(* IEC 61131-3 sources: Livny/, 3 files *)

(* ---- 03_FB_InputHandler.st ---- *)
(* =========================================================================
   ПРОЕКТ    : Весовой дозатор сахара в мешки 25/50 кг («Ливны»)
   ПЛАТФОРМА : ОВЕН СПК107 · CODESYS 3.5.17 · IEC 61131-3 (Structured Text)
   =========================================================================
   ФАЙЛ      : 03_FB_InputHandler.st
   НАЗНАЧЕНИЕ: Антидребезг дискретных входов (МВ110-8Д.4Р) и выделение
               фронтов кнопок. Дискретизация опроса модуля по RS-485 —
               десятки мс, поэтому фильтруем 40 мс (TON).

               В CODESYS: "Добавить объект → ФБ", язык ST.
   ========================================================================= *)

FUNCTION_BLOCK FB_InputHandler

VAR_INPUT
    xRawStart       : BOOL;   (* «сырой» DI0 ПУСК                         *)
    xRawStop        : BOOL;   (* «сырой» DI1 СТОП                         *)
    xRawEStop       : BOOL;   (* «сырой» DI2 АВАРИЙНЫЙ СТОП (НЗ-контакт)  *)
    xRawBag         : BOOL;   (* «сырой» DI3 мешок в зоне                 *)
    xRawClampClosed : BOOL;   (* «сырой» DI4 концевик зажима              *)
    xRawAirOK       : BOOL;   (* «сырой» DI5 давление воздуха             *)
    xRawLevel       : BOOL;   (* «сырой» DI6 уровень в бункере            *)
    xRawCover       : BOOL;   (* «сырой» DI7 защитная крышка              *)
END_VAR

VAR_OUTPUT
    xStart        : BOOL;     (* ПУСК, отфильтрованный                    *)
    xStop         : BOOL;     (* СТОП, отфильтрованный                    *)
    xStartUp      : BOOL;     (* фронт кнопки ПУСК (один скан)            *)
    xStopUp       : BOOL;     (* фронт кнопки СТОП (один скан)            *)
    xEStop        : BOOL;     (* АВАРИЯ активна (инверсия НЗ-контакта)    *)
    xBagPresent   : BOOL;     (* мешок установлен в зону загрузки         *)
    xClampClosed  : BOOL;     (* зажим механически закрыт                 *)
    xAirOK        : BOOL;     (* давление пневмосети в норме              *)
    xLevelOK      : BOOL;     (* продукт в бункере есть                   *)
    xCoverClosed  : BOOL;     (* защитная крышка закрыта                  *)
END_VAR

VAR
    (* Фильтры антидребезга: TON с выдержкой tDebounce                  *)
    tonStart : TON;
    tonStop  : TON;
    tonEStop : TON;
    tonBag   : TON;
    tonClamp : TON;
    tonAir   : TON;
    tonLevel : TON;
    tonCover : TON;

    (* Детекторы фронта для кнопок                                      *)
    rtStart  : R_TRIG;
    rtStop   : R_TRIG;

    tDebounce : TIME := T#40MS;  (* Постоянная антидребезга               *)
END_VAR

(* ---------------------------------------------------------------------
   1. АНТИДРЕБЕЗГ. Вход считается принятым, если удерживается
      не менее tDebounce. Для цепей безопасности (аварийный стоп)
      это не ухудшает быстродействие: НЗ-контакт при срабатывании
      РАЗМЫКАЕТСЯ, и инверсный признак аварии снимает разрешение
      выходов уже в следующем скане.
   --------------------------------------------------------------------- *)
tonStart(IN := xRawStart,       PT := tDebounce);
tonStop (IN := xRawStop,        PT := tDebounce);
tonEStop(IN := xRawEStop,       PT := tDebounce);
tonBag  (IN := xRawBag,         PT := tDebounce);
tonClamp(IN := xRawClampClosed, PT := tDebounce);
tonAir  (IN := xRawAirOK,       PT := tDebounce);
tonLevel(IN := xRawLevel,       PT := tDebounce);
tonCover(IN := xRawCover,       PT := tDebounce);

xStart       := tonStart.Q;
xStop        := tonStop.Q;

(* Аварийный стоп — НЗ-контакт: пока цепь цела, вход = TRUE.
   Размыкание (нажатие/обрыв) даёт xEStop = TRUE.                     *)
xEStop       := NOT tonEStop.Q;

xBagPresent  := tonBag.Q;
xClampClosed := tonClamp.Q;
xAirOK       := tonAir.Q;
xLevelOK     := tonLevel.Q;
xCoverClosed := tonCover.Q;

(* ---------------------------------------------------------------------
   2. ФРОНТЫ КНОПОК — для запуска/останова цикла из любого состояния.
   --------------------------------------------------------------------- *)
rtStart(CLK := xStart);
xStartUp := rtStart.Q;

rtStop(CLK := xStop);
xStopUp  := rtStop.Q;

END_FUNCTION_BLOCK

(* =========================================================================
   КОНЕЦ ФАЙЛА 03_FB_InputHandler.st
   ========================================================================= *)

(* ---- 05_FB_DoserControl.st ---- *)
(* =========================================================================
   ПРОЕКТ    : Весовой дозатор сахара в мешки 25/50 кг («Ливны»)
   ПЛАТФОРМА : ОВЕН СПК107 · CODESYS 3.5.17 · IEC 61131-3 (Structured Text)
   =========================================================================
   ФАЙЛ      : 05_FB_DoserControl.st
   НАЗНАЧЕНИЕ: Управляющий автомат дозатора (ядро проекта).

   ЦИКЛ ДОЗИРОВАНИЯ:
     ГОТОВНОСТЬ → ЗАЖИМ → ТАРА → ГРУБАЯ ПОДАЧА → ТОЧНАЯ ПОДАЧА →
     УСПОКОЕНИЕ → КОНТРОЛЬ (→ ДОСЫПКА) → СБРОС МЕШКА → ПАУЗА → ГОТОВНОСТЬ

   КЛЮЧЕВЫЕ ПРИНЦИПЫ:
     1. Двухступенчатая подача: основной шнек даёт ~90 % дозы,
        малый шнек — доводка. Это главный способ получить точность
        ±50 г на мешке 25 кг при грубой пневматике/механике.
     2. Отсечка «на лету» (in-flight): питатель закрывается ДО
        достижения уставки на величину продукта, который ещё летит
        в мешок:  W_отс = W_зад − Δ_лету.
     3. Адаптация Δ_лету по ошибке каждой отвешенной дозы:
        ε = W_факт − W_зад ≈ Δ_факт − Δ_принято
        Δ_лету := clamp( Δ_лету + K·ε ,  Δ_min … Δ_max )
     4. Контроль потока: за окно tFlowCheck вес обязан вырасти
        не менее чем на rFlowMinStep — иначе «затор/пусто».
     5. Failsafe: при любой аварии выходы гасятся в том же скане.
   ========================================================================= *)

FUNCTION_BLOCK FB_DoserControl

VAR_INPUT
    xEnable      : BOOL;   (* разрешение работы автоматики               *)
    xAlarmActive : BOOL;   (* есть квитируемые аварии (от FB_AlarmManager)*)
    xStartCmd    : BOOL;   (* импульс «ПУСК» (один скан)                 *)
    xStopCmd     : BOOL;   (* импульс «СТОП» (один скан)                 *)
    xAckCmd      : BOOL;   (* импульс квитирования                       *)

    (* Весовой канал (после FB_WeightChannel)                           *)
    rNet     : REAL;       (* вес нетто, кг                              *)
    xStable  : BOOL;       (* вес стабилен                               *)
    xCommOK  : BOOL;       (* связь с тензомодулем в норме               *)

    (* Дискретные сигналы (после FB_InputHandler)                       *)
    xBagPresent   : BOOL;  (* мешок в зоне загрузки                      *)
    xClampClosed  : BOOL;  (* концевик: зажим закрыт                     *)
    xAirOK        : BOOL;  (* давление пневмосети в норме                *)
    xLevelOK      : BOOL;  (* сахар в расходном бункере есть             *)
    xCoverClosed  : BOOL;  (* защитная крышка закрыта                    *)
    xEStop        : BOOL;  (* аварийный стоп (НЗ-цепь)                   *)

    (* Технологические параметры                                        *)
    p : ST_DoseParams;
END_VAR

VAR_OUTPUT
    xDoClamp  : BOOL;      (* пневмоклапан зажима мешка                  *)
    xDoCoarse : BOOL;      (* грубый питатель (основной шнек)            *)
    xDoFine   : BOOL;      (* точный питатель (малый шнек)               *)
    xTareReq  : BOOL;      (* импульс тарирования → FB_WeightChannel     *)

    eState    : E_DoserState;   (* текущее состояние (для HMI/архива)    *)
    rInFlight : REAL;           (* текущая адаптивная отсечка, кг        *)
    rLastError: REAL;           (* ошибка последней дозы, кг             *)

    (* Запросы на аварии (защёлкиваются в FB_AlarmManager)              *)
    xReqTareFault : BOOL;
    xReqNoFlow    : BOOL;
    xReqOverdose  : BOOL;
    xReqUnderdose : BOOL;
    xReqClamp     : BOOL;
END_VAR

VAR_IN_OUT
    stStats : ST_DoseStats;    (* статистика смены (хранится в GVL)      *)
END_VAR

VAR
    ePrev      : E_DoserState := ST_STOP;
    xEntry     : BOOL;         (* первый скан в состоянии               *)
    xTareSent  : BOOL;         (* импульс тарирования уже выдан         *)

    tonClamp   : TON;          (* контроль закрытия зажима              *)
    tonTare    : TON;          (* контроль времени тарирования          *)
    tonSettle  : TON;          (* успокоение продукта                   *)
    tonFlow    : TON;          (* окно контроля потока (самоперезапуск) *)
    tonTopup   : TON;          (* ограничение времени досыпки           *)
    tonRelease : TON;          (* время разжима                         *)
    tonPause   : TON;          (* пауза между циклами                   *)

    rFlowBase  : REAL;         (* вес в начале окна контроля потока     *)
    rInFlightI : REAL;         (* внутренняя адаптивная отсечка, кг     *)
    rSnapshot  : REAL;         (* вес после успокоения, кг              *)
    rErr       : REAL;         (* ошибка дозы, кг                       *)
    rBagWeight : REAL;         (* вес пустого мешка при тарировании, кг *)
    iTopupCnt  : INT;          (* счётчик попыток досыпки               *)
    xInitDone  : BOOL;
END_VAR

(* ---------------------------------------------------------------------
   0. ИНИЦИАЛИЗАЦИЯ И ОБЩИЕ ПРАВИЛА
   --------------------------------------------------------------------- *)
IF NOT xInitDone THEN
    rInFlightI := p.rInFlightInit;   (* стартовая оценка отсечки       *)
    xInitDone  := TRUE;
END_IF

rInFlight := rInFlightI;             (* наружу — для HMI/трендов       *)

(* Безопасные выходы по умолчанию. Каждый шаг сам «поднимает»
   нужные выходы — при любом сбое шаг не отрабатывается => всё отключено. *)
xDoClamp  := FALSE;
xDoCoarse := FALSE;
xDoFine   := FALSE;
xTareReq  := FALSE;

(* Жёсткая авария: аварийный стоп или потеря весов — мгновенно.        *)
IF (xEStop OR NOT xCommOK) AND (eState <> ST_STOP) AND (eState <> ST_ALARM) THEN
    eState := ST_ALARM;
END_IF

(* Запрет автоматики (например, включён РУЧНОЙ режим) → в ОСТАНОВ.    *)
IF NOT xEnable AND (eState <> ST_STOP) AND (eState <> ST_ALARM) THEN
    eState := ST_STOP;
END_IF

(* Таймеры по умолчанию сброшены; используемые шаги взводят IN.        *)
tonClamp(IN := FALSE);
tonTare(IN := FALSE);
tonSettle(IN := FALSE);
tonFlow(IN := FALSE);
tonTopup(IN := FALSE);
tonRelease(IN := FALSE);
tonPause(IN := FALSE);

(* Флаг входа в состояние — для одноразовых действий.                  *)
xEntry := (eState <> ePrev);

(* ---------------------------------------------------------------------
   1. АВТОМАТ СОСТОЯНИЙ
   --------------------------------------------------------------------- *)
CASE eState OF

    (* ── ОСТАНОВ ─────────────────────────────────────────────────── *)
    ST_STOP:
        IF xEnable AND NOT xAlarmActive THEN
            eState := ST_READY;
        END_IF

    (* ── ГОТОВНОСТЬ: ждём ПУСК и проверяем разрешения ────────────── *)
    ST_READY:
        IF xStartCmd
           AND xBagPresent AND xAirOK AND xLevelOK AND xCoverClosed
           AND NOT xAlarmActive THEN
            iTopupCnt := 0;
            eState    := ST_CLAMPING;
        END_IF

    (* ── ЗАЖИМ МЕШКА ─────────────────────────────────────────────── *)
    ST_CLAMPING:
        xDoClamp := TRUE;
        tonClamp(IN := TRUE, PT := p.tClampTimeout);
        IF xClampClosed THEN
            eState := ST_TARE;                (* концевик подтвердил   *)
        ELSIF tonClamp.Q THEN
            xReqClamp := TRUE;                (* зажим не закрылся     *)
            eState    := ST_ALARM;
        END_IF

    (* ── ТАРИРОВАНИЕ ─────────────────────────────────────────────── *)
    ST_TARE:
        xDoClamp := TRUE;

        IF xEntry THEN
            rBagWeight := rNet;               (* сейчас на весах только мешок *)
            xTareSent  := FALSE;
            (* правдоподобие веса пустого мешка *)
            IF (rBagWeight < p.rTareMin) OR (rBagWeight > p.rTareMax) THEN
                xReqTareFault := TRUE;        (* нет мешка / посторонний груз *)
                eState        := ST_ALARM;
            END_IF
        END_IF

        (* импульс тарирования — один раз, когда вес стабилен *)
        IF (eState = ST_TARE) AND xStable AND NOT xTareSent THEN
            xTareReq  := TRUE;                (* → FB_WeightChannel    *)
            xTareSent := TRUE;
        END_IF

        tonTare(IN := TRUE, PT := p.tTareTimeout);
        IF xTareSent AND ABS(rNet) <= p.rStabBand THEN
            eState := ST_FEED_COARSE;         (* ноль установлен       *)
        ELSIF tonTare.Q THEN
            xReqTareFault := TRUE;            (* не удалось стабилизировать *)
            eState        := ST_ALARM;
        END_IF

    (* ── ГРУБАЯ ПОДАЧА (~90 % дозы) ──────────────────────────────── *)
    ST_FEED_COARSE:
        xDoClamp  := TRUE;
        xDoCoarse := TRUE;

        IF xEntry THEN
            rFlowBase := rNet;
        END_IF

        (* контроль потока: самоперезапускающееся окно tFlowCheck *)
        tonFlow(IN := NOT tonFlow.Q, PT := p.tFlowCheck);
        IF tonFlow.Q THEN
            IF (rNet - rFlowBase) < p.rFlowMinStep THEN
                xReqNoFlow := TRUE;           (* затор шнека / пусто   *)
                eState     := ST_ALARM;
            ELSE
                rFlowBase := rNet;            (* следующее окно        *)
            END_IF
        END_IF

        (* отсечка грубой подачи *)
        IF rNet >= (p.rSetpoint - p.rCoarseCutoff) THEN
            eState := ST_FEED_FINE;
        END_IF

    (* ── ТОЧНАЯ ПОДАЧА (доводка малым шнеком) ────────────────────── *)
    ST_FEED_FINE:
        xDoClamp := TRUE;
        xDoFine  := TRUE;

        IF xEntry THEN
            rFlowBase := rNet;
        END_IF

        (* контроль потока (порог ниже — подача медленная) *)
        tonFlow(IN := NOT tonFlow.Q, PT := p.tFlowCheck);
        IF tonFlow.Q THEN
            IF (rNet - rFlowBase) < p.rFineFlowMin THEN
                xReqNoFlow := TRUE;
                eState     := ST_ALARM;
            ELSE
                rFlowBase := rNet;
            END_IF
        END_IF

        (* отсечка «на лету» с адаптивной поправкой *)
        IF rNet >= (p.rSetpoint - rInFlightI) THEN
            eState := ST_SETTLING;
        END_IF

    (* ── УСПОКОЕНИЕ: продукт досыпается, вес стабилизируется ─────── *)
    ST_SETTLING:
        xDoClamp := TRUE;
        tonSettle(IN := TRUE, PT := p.tSettle);
        IF tonSettle.Q THEN
            rSnapshot := rNet;                (* фиксируем результат   *)
            eState    := ST_CHECK;
        END_IF

    (* ── КОНТРОЛЬ ДОЗЫ И ОБУЧЕНИЕ ────────────────────────────────── *)
    ST_CHECK:
        xDoClamp := TRUE;
        rErr       := rSnapshot - p.rSetpoint;
        rLastError := rErr;

        IF rErr > p.rTolerancePlus THEN
            (* ПЕРЕДОЗ: автоматически высыпать нельзя — зовём оператора *)
            stStats.diOver := stStats.diOver + 1;
            xReqOverdose   := TRUE;
            eState         := ST_ALARM;

        ELSIF rErr < -p.rToleranceMinus THEN
            (* НЕДОВЕС: пробуем досыпать малым шнеком *)
            IF iTopupCnt < p.iTopupMax THEN
                eState := ST_TOPUP;
            ELSE
                stStats.diUnder := stStats.diUnder + 1;
                xReqUnderdose   := TRUE;
                eState          := ST_ALARM;
            END_IF

        ELSE
            (* ДОЗА В ДОПУСКЕ — адаптация и статистика *)
            IF p.xLearnEnable THEN
                (* Δ_лету := clamp( Δ_лету + K·ε ,  Δ_min … Δ_max ) *)
                rInFlightI := LIMIT(p.rInFlightMin,
                                    rInFlightI + p.rLearnGain * rErr,
                                    p.rInFlightMax);
            END_IF

            stStats.diCount    := stStats.diCount + 1;
            stStats.rLastNet   := rSnapshot;
            stStats.rLastError := rErr;
            stStats.rTotalNet  := stStats.rTotalNet + rSnapshot;
            stStats.rSumError  := stStats.rSumError + rErr;

            IF stStats.diCount = 1 THEN
                stStats.rMinNet := rSnapshot;
                stStats.rMaxNet := rSnapshot;
            ELSE
                stStats.rMinNet := MIN(stStats.rMinNet, rSnapshot);
                stStats.rMaxNet := MAX(stStats.rMaxNet, rSnapshot);
            END_IF

            eState := ST_UNCLAMP;
        END_IF

    (* ── ДОСЫПКА ПРИ НЕДОВЕСЕ ────────────────────────────────────── *)
    ST_TOPUP:
        xDoClamp := TRUE;
        xDoFine  := TRUE;

        IF xEntry THEN
            iTopupCnt        := iTopupCnt + 1;
            stStats.diTopups := stStats.diTopups + 1;
        END_IF

        tonTopup(IN := TRUE, PT := p.tTopupMax);
        IF (rNet >= (p.rSetpoint - rInFlightI)) OR tonTopup.Q THEN
            eState := ST_SETTLING;            (* снова успокоение+контроль *)
        END_IF

    (* ── СБРОС МЕШКА ─────────────────────────────────────────────── *)
    ST_UNCLAMP:
        xDoClamp := FALSE;                    (* разжим — мешок уходит *)
        tonRelease(IN := TRUE, PT := p.tRelease);
        IF tonRelease.Q THEN
            eState := ST_PAUSE;
        END_IF

    (* ── ПАУЗА ПЕРЕД СЛЕДУЮЩИМ ЦИКЛОМ ────────────────────────────── *)
    ST_PAUSE:
        tonPause(IN := TRUE, PT := p.tPause);
        IF tonPause.Q THEN
            eState := ST_READY;
        END_IF

    (* ── АВАРИЯ: выходы погашены, ждём квитирования ──────────────── *)
    ST_ALARM:
        IF xAckCmd AND NOT xAlarmActive AND NOT xEStop AND xCommOK THEN
            eState := ST_STOP;                (* квитировано → перезапуск *)
        END_IF

END_CASE

(* ---------------------------------------------------------------------
   2. ОПЕРАТИВНЫЙ «СТОП» ИЗ ЛЮБОГО РАБОЧЕГО СОСТОЯНИЯ:
      подача останавливается, мешок сбрасывается — безопасный выход.
   --------------------------------------------------------------------- *)
IF xStopCmd AND (eState <> ST_STOP) AND (eState <> ST_ALARM) THEN
    eState := ST_UNCLAMP;
END_IF

(* Запомнить состояние для флага xEntry следующего скана.              *)
ePrev := eState;

END_FUNCTION_BLOCK

(* =========================================================================
   КОНЕЦ ФАЙЛА 05_FB_DoserControl.st
   ========================================================================= *)

(* ---- 07_PRG_Main.st ---- *)
(* =========================================================================
   ПРОЕКТ    : Весовой дозатор сахара в мешки 25/50 кг («Ливны»)
   ПЛАТФОРМА : ОВЕН СПК107 · CODESYS 3.5.17 · IEC 61131-3 (Structured Text)
   =========================================================================
   ФАЙЛ      : 07_PRG_Main.st
   НАЗНАЧЕНИЕ: Главная программа (PRG). Собирает контур управления:
               FB_InputHandler → FB_WeightChannel → FB_DoserControl
               → FB_AlarmManager, плюс режим РУЧНОЙ для пусконаладки.

               Размещается в основной задаче СПК107 (цикл 10…20 мс).
   ========================================================================= *)

PROGRAM PRG_Main

VAR
    fbIn   : FB_InputHandler;   (* антидребезг входов                    *)
    fbW    : FB_WeightChannel;  (* весовой канал                         *)
    fbDose : FB_DoserControl;   (* автомат дозирования                   *)
    fbAlm  : FB_AlarmManager;   (* аварии                                *)

    (* Фронты экранных кнопок СПК107 *)
    rtHmiStart : R_TRIG;
    rtHmiStop  : R_TRIG;
    rtHmiAck   : R_TRIG;
    rtHmiTare  : R_TRIG;

    xCmdStart : BOOL;   (* объединённый ПУСК: кнопка на щите ИЛИ экран  *)
    xCmdStop  : BOOL;   (* объединённый СТОП                            *)
    xCmdAck   : BOOL;   (* объединённое квитирование                    *)
END_VAR

(* ---------------------------------------------------------------------
   1. ОБРАБОТКА ДИСКРЕТНЫХ ВХОДОВ (антидребезг 40 мс, фронты кнопок)
   --------------------------------------------------------------------- *)
fbIn(
    xRawStart       := g_xDiStart,
    xRawStop        := g_xDiStop,
    xRawEStop       := g_xDiEStop,
    xRawBag         := g_xDiBagPresent,
    xRawClampClosed := g_xDiClampClosed,
    xRawAirOK       := g_xDiAirOK,
    xRawLevel       := g_xDiLevelOK,
    xRawCover       := g_xDiCoverClosed
);

(* ---------------------------------------------------------------------
   2. КОМАНДЫ УПРАВЛЕНИЯ: аппаратные кнопки + экран СПК107
   --------------------------------------------------------------------- *)
rtHmiStart(CLK := g_xHmiStart);
rtHmiStop (CLK := g_xHmiStop);
rtHmiAck  (CLK := g_xHmiAck);
rtHmiTare (CLK := g_xHmiTare);

xCmdStart := fbIn.xStartUp OR rtHmiStart.Q;
xCmdStop  := fbIn.xStopUp  OR rtHmiStop.Q;
xCmdAck   := rtHmiAck.Q;

(* ---------------------------------------------------------------------
   3. ВЕСОВОЙ КАНАЛ (фильтр, стабильность, тара, скорость потока)
   --------------------------------------------------------------------- *)
fbW(
    rWeightRaw  := g_rWeightRaw,
    xValid      := g_xWeightValid,
    xError      := g_xWeightErr,
    xTareCmd    := fbDose.xTareReq,
    xTareManual := rtHmiTare.Q OR g_Manual.xTare,
    rStabBand   := g_Params.rStabBand,
    tStabTime   := g_Params.tStabTime
);

(* обработанные данные — в глобальную структуру *)
g_Weight.rNet      := fbW.rNet;
g_Weight.rGross    := fbW.rGross;
g_Weight.rTare     := fbW.rTare;
g_Weight.xStable   := fbW.xStable;
g_Weight.rFlowRate := fbW.rFlowRate;
g_Weight.xCommOK   := fbW.xCommOK;

(* аппаратная установка нуля в МВ110-224.1ТД *)
g_xTareToModule := fbW.xTarePulse;

(* ---------------------------------------------------------------------
   4. УПРАВЛЕНИЕ: АВТОМАТ ИЛИ РУЧНОЙ РЕЖИМ
   --------------------------------------------------------------------- *)
IF g_xManualMode THEN
    (* РУЧНОЙ РЕЖИМ (пусконаладка/обслуживание):
       прямое управление выходами с экрана, с аппаратными блокировками. *)
    g_xDoClamp  := g_Manual.xClamp  AND fbIn.xAirOK AND NOT fbIn.xEStop;
    g_xDoCoarse := g_Manual.xCoarse AND NOT fbIn.xEStop AND fbIn.xCoverClosed;
    g_xDoFine   := g_Manual.xFine   AND NOT fbIn.xEStop AND fbIn.xCoverClosed;
    g_xDoSignal := g_Manual.xSignal;
    g_eState    := ST_STOP;               (* автомат остановлен       *)

ELSE
    (* АВТОМАТИЧЕСКИЙ РЕЖИМ *)
    fbDose(
        xEnable      := NOT g_xManualMode,
        xAlarmActive := fbAlm.xActiveAny,
        xStartCmd    := xCmdStart,
        xStopCmd     := xCmdStop,
        xAckCmd      := xCmdAck,

        rNet    := fbW.rNet,
        xStable := fbW.xStable,
        xCommOK := fbW.xCommOK,

        xBagPresent  := fbIn.xBagPresent,
        xClampClosed := fbIn.xClampClosed,
        xAirOK       := fbIn.xAirOK,
        xLevelOK     := fbIn.xLevelOK,
        xCoverClosed := fbIn.xCoverClosed,
        xEStop       := fbIn.xEStop,

        p       := g_Params,
        stStats := g_Stats
    );

    g_xDoClamp  := fbDose.xDoClamp;
    g_xDoCoarse := fbDose.xDoCoarse;
    g_xDoFine   := fbDose.xDoFine;
    g_eState    := fbDose.eState;
END_IF

(* ---------------------------------------------------------------------
   5. АВАРИИ: сбор запросов, защёлкивание, мигалка
   --------------------------------------------------------------------- *)
fbAlm(
    xEStop         := fbIn.xEStop,
    xCommLoss      := NOT fbW.xCommOK,
    xAirOK         := fbIn.xAirOK,
    xLevelOK       := fbIn.xLevelOK,
    xCoverClosed   := fbIn.xCoverClosed,
    xReqTareFault  := fbDose.xReqTareFault,
    xReqNoFlow     := fbDose.xReqNoFlow,
    xReqOverdose   := fbDose.xReqOverdose,
    xReqUnderdose  := fbDose.xReqUnderdose,
    xReqClamp      := fbDose.xReqClamp,
    xAckAll        := xCmdAck
);

g_Alarms := fbAlm.stA;

(* ---------------------------------------------------------------------
   6. СИГНАЛЬНАЯ ЛАМПА (в авто-режиме):
      авария — мигание 1 Гц; дозирование — ровный свет; простой — выкл.
   --------------------------------------------------------------------- *)
IF NOT g_xManualMode THEN
    IF g_Alarms.xActive THEN
        g_xDoSignal := fbAlm.xLampBlink;
    ELSIF (g_eState <> ST_STOP) AND (g_eState <> ST_READY) THEN
        g_xDoSignal := TRUE;
    ELSE
        g_xDoSignal := FALSE;
    END_IF
END_IF

END_PROGRAM

(* =========================================================================
   КОНЕЦ ФАЙЛА 07_PRG_Main.st
   ========================================================================= *)
